// TwinCAT 3 PLC project PLC_AtoB_PlantCtrl
// ProgramVersion: 3.1.4024.0
// libraries:
//   Tc2_Standard, * (Beckhoff Automation GmbH)
//   Tc2_System, * (Beckhoff Automation GmbH)
//   Tc3_Module, * (Beckhoff Automation GmbH)
// project tree:
//   DUTs/ Udt_CM_Actuator3State.TcDUT, Udt_CM_Sensor2State.TcDUT, Udt_PlantControl_Out.TcDUT
//   GVLs/ FIO.TcGVL
//   / PlcTask.TcTTO
//   POUs/CMs/ CM_Actuator3State.TcPOU, CM_Sensor2State.TcPOU
//   POUs/ FB_PlantControl.TcPOU, MAIN.TcPOU, Prg_StateMachine.TcPOU
// real-time tasks:
//   TASK PlcTask: cycle T#10ms, priority 20, ADS port 350

CONFIGURATION PLC_AtoB_PlantCtrl
    RESOURCE PLC ON TwinCAT3
        TASK PlcTask(INTERVAL := T#10ms, PRIORITY := 20);
        PROGRAM MAIN WITH PlcTask : MAIN;
    END_RESOURCE
END_CONFIGURATION

// ---- DUTs/Udt_CM_Actuator3State.TcDUT
TYPE Udt_CM_Actuator3State :
STRUCT
	output_state1 : BOOL;
	output_state2 : BOOL;
	output_state3 : BOOL;
	
END_STRUCT
END_TYPE

// ---- DUTs/Udt_CM_Sensor2State.TcDUT
TYPE Udt_CM_Sensor2State :
STRUCT
	sensor_Input : BOOL;
	
	sensor_Output : BOOL; 
END_STRUCT
END_TYPE

// ---- DUTs/Udt_PlantControl_Out.TcDUT
TYPE Udt_PlantControl_Out :
STRUCT
	Auto_Out : BOOL;
	Manual_Out : BOOL;
	
	Startet_Out : BOOL;
	Stopped_Out : BOOL;
	Reset_Out : BOOL;
	ResetEmgStop_Out_5s :BOOL;
	
	EmgStopped_Out : BOOL;
END_STRUCT
END_TYPE

// ---- GVLs/FIO.TcGVL
{attribute 'qualified_only'}
VAR_GLOBAL
	
	bEmgStop : BOOL := TRUE; //Sensor	Bool	Emergency stop	0	TRUE
	bStart : BOOL;	//Sensor	Bool	Start	1	FALSE
	bStop : BOOL := TRUE;	//Sensor	Bool	Stop	3	TRUE
	bReset : BOOL;	//Sensor	Bool	Reset	4	FALSE
	bManual : BOOL;	//Sensor	Bool	Manual	5	TRUE
	bAuto : BOOL; 	//Sensor	Bool	Auto	6	FALSE
	
	bGreenLight : BOOL;
	bYellowLight : BOOL;
	bRedLight : BOOL;
	
	
	bSensorB : BOOL;
	bSensorA : BOOL;
	
	bEntryConveyor : BOOL;
	
	bConveyorCW : BOOL;
	bConveyorCCW : BOOL;
//Sensor	Bool	Sensor B	1	TRUE
//Sensor	Bool	Sensor A	0	TRUE

//Actuator	Bool	Roller Conveyor (4m) 1 (+)	0	FALSE
//Actuator	Bool	Roller Conveyor (4m) 1 (-)	2	FALSE
//Actuator	Bool	Entry conveyor	1	FALSE



END_VAR

// ---- POUs/MAIN.TcPOU
PROGRAM MAIN
VAR
	fbPlantControl : FB_PlantControl;
	Ctrl_data_Plant : Udt_PlantControl_Out;
	
	Ctrl_data_StateMachine :Udt_PlantControl_Out;
	
	cmSensorA : CM_Sensor2State;
	Ctrl_data_SensorA : Udt_CM_Sensor2State;
	
	cmSensorB : CM_Sensor2State;
	Ctrl_data_SensorB : Udt_CM_Sensor2State;
	
	cmConveyorEntry : CM_Actuator3State;
	Ctrl_data_ConveyorEntry : Udt_CM_Actuator3State;
	
	cmConveyorMain : CM_Actuator3State;
	Ctrl_data_ConveyorMain : Udt_CM_Actuator3State;
END_VAR

fbPlantControl(
	//Set up variables to IO here
	Auto_In := FIO.bAuto,
	Manual_In := FIO.bManual,
	
	Start_In := FIO.bStart,
	Stop_In := FIO.bStop,
	EmgStop_In := FIO.bEmgStop,
	Reset_In := FIO.bReset,
	
	Startet_Out => FIO.bGreenLight,
	Stopped_Out => FIO.bYellowLight,
	EmgStopped_Out => FIO.bRedLight,

	Ctrl_Plant := Ctrl_data_Plant
	);
	
Prg_StateMachine(
	Plant_Ctrl := Ctrl_data_Plant,
	
	cmSensor2State_sensorA := Ctrl_data_SensorA,
	cmSensor2State_sensorB := Ctrl_data_SensorB,

	cmActuator3State_ConveyorEntry :=  Ctrl_data_ConveyorEntry,
	cmActuator3State_ConveyorMain := Ctrl_data_ConveyorMain
);

cmSensorA(
	sensorInput := FIO.bSensorA,

	Ctrl_CM_Sensor2State := Ctrl_data_SensorA
	);
cmSensorB(
	sensorInput := FIO.bSensorB,

	Ctrl_CM_Sensor2State := Ctrl_data_SensorB
	);
	
cmConveyorEntry(
	output_2 => FIO.bEntryConveyor,
	
	Ctrl_CM_Actuator3State := Ctrl_data_ConveyorEntry
	);
	
cmConveyorMain(
	output_2 => FIO.bConveyorCW,
	output_3 => FIO.bConveyorCCW,
	
	Ctrl_CM_Actuator3State := Ctrl_data_ConveyorMain
	);

END_PROGRAM

// ---- POUs/FB_PlantControl.TcPOU
FUNCTION_BLOCK FB_PlantControl
VAR_INPUT
	Auto_In : BOOL;
	Manual_In : BOOL;
	
	Start_In : BOOL;
	Stop_In : BOOL;
	Reset_In : BOOL;
	
	EmgStop_In : BOOL;
	
END_VAR
VAR_OUTPUT
	Auto_Out : BOOL;
	Manual_Out : BOOL;
	
	Startet_Out : BOOL;
	Stopped_Out : BOOL;
	Reset_Out : BOOL;
	ResetEmgStop_Out_5s :BOOL;
	
	EmgStopped_Out : BOOL;
END_VAR
VAR
END_VAR
VAR_IN_OUT
	Ctrl_Plant : Udt_PlantControl_Out;
END_VAR

VAR CONSTANT
	SR_Auto: SR;
	SR_Man : SR;
	
	SR_start : SR;
	SR_Stop : SR;
	
	EmgResetTimerOff : Tc2_Standard.TON;
END_VAR

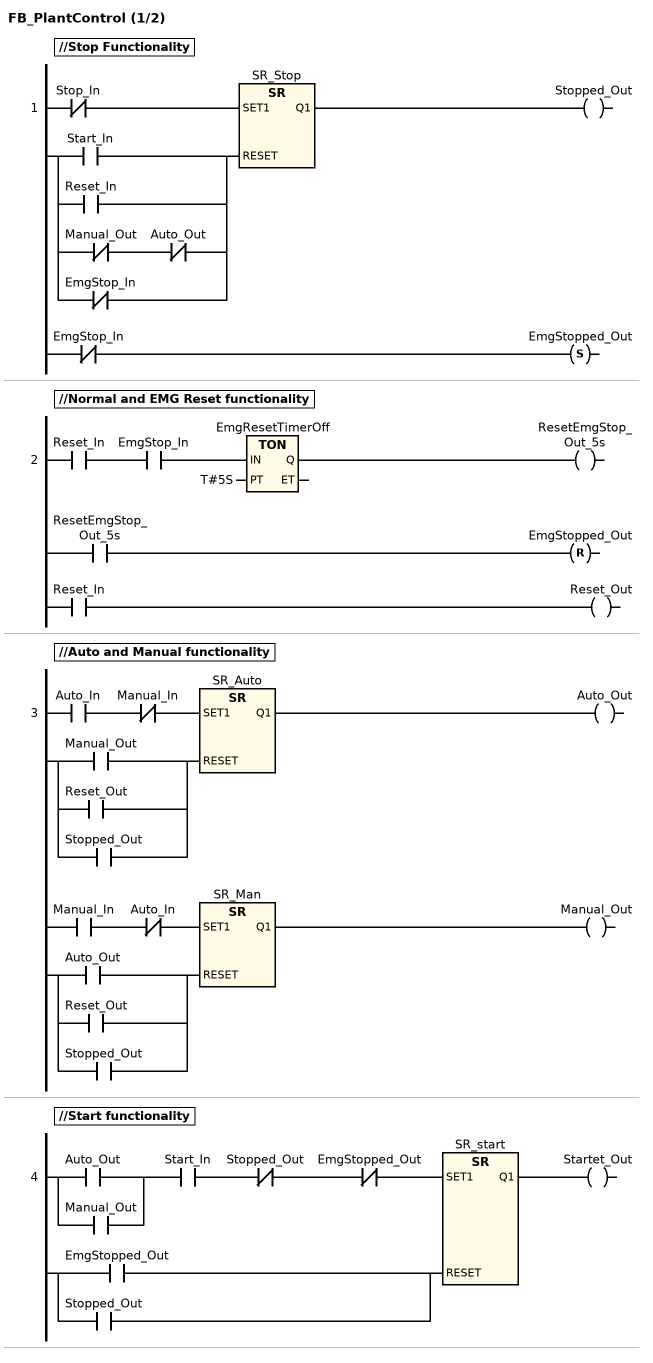
// NETWORK 1
// label: //Stop Functionality
SR_Stop(SET1 := NOT Stop_In, RESET := Start_In OR Reset_In OR NOT Manual_Out AND NOT Auto_Out OR NOT EmgStop_In); // SR
Stopped_Out := SR_Stop.Q1;
EmgStopped_Out S= NOT EmgStop_In;

// NETWORK 2
// label: //Normal and EMG Reset functionality
EmgResetTimerOff(IN := Reset_In AND EmgStop_In, PT := T#5S); // TON
ResetEmgStop_Out_5s := EmgResetTimerOff.Q;
EmgStopped_Out R= ResetEmgStop_Out_5s;
Reset_Out := Reset_In;

// NETWORK 3
// label: //Auto and Manual functionality
SR_Auto(SET1 := Auto_In AND NOT Manual_In, RESET := Manual_Out OR Reset_Out OR Stopped_Out); // SR
Auto_Out := SR_Auto.Q1;
SR_Man(SET1 := Manual_In AND NOT Auto_In, RESET := Auto_Out OR Reset_Out OR Stopped_Out); // SR
Manual_Out := SR_Man.Q1;

// NETWORK 4
// label: //Start functionality
SR_start(SET1 := (Auto_Out OR Manual_Out) AND Start_In AND NOT Stopped_Out AND NOT EmgStopped_Out, RESET := EmgStopped_Out OR Stopped_Out); // SR
Startet_Out := SR_start.Q1;

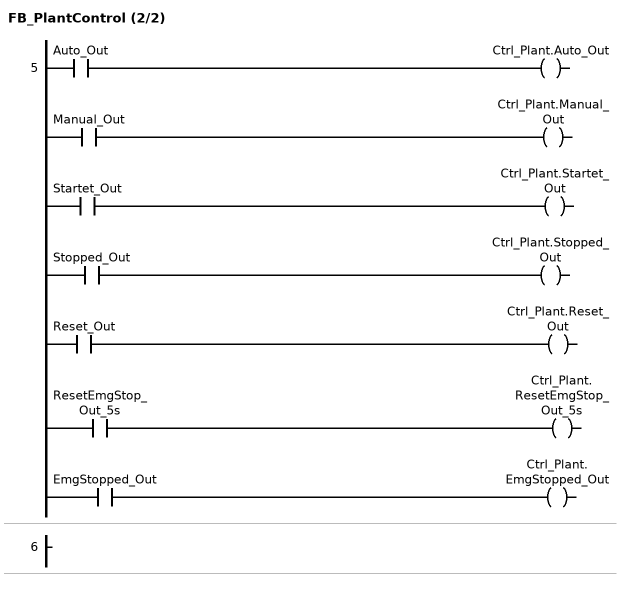
// NETWORK 5
Ctrl_Plant.Auto_Out := Auto_Out;
Ctrl_Plant.Manual_Out := Manual_Out;
Ctrl_Plant.Startet_Out := Startet_Out;
Ctrl_Plant.Stopped_Out := Stopped_Out;
Ctrl_Plant.Reset_Out := Reset_Out;
Ctrl_Plant.ResetEmgStop_Out_5s := ResetEmgStop_Out_5s;
Ctrl_Plant.EmgStopped_Out := EmgStopped_Out;

// NETWORK 6

END_FUNCTION_BLOCK

// ---- POUs/CMs/CM_Sensor2State.TcPOU
FUNCTION_BLOCK CM_Sensor2State
VAR_INPUT
	sensorInput : BOOL;
END_VAR
VAR_OUTPUT
	sensoroutput : BOOL;
END_VAR
VAR_IN_OUT
	Ctrl_CM_Sensor2State : Udt_CM_Sensor2State; 
END_VAR
VAR
END_VAR

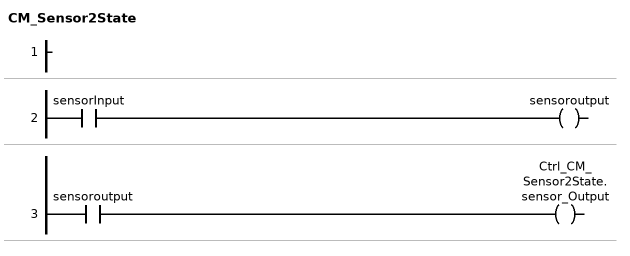
// NETWORK 1

// NETWORK 2
sensoroutput := sensorInput;

// NETWORK 3
Ctrl_CM_Sensor2State.sensor_Output := sensoroutput;

END_FUNCTION_BLOCK

// ---- POUs/CMs/CM_Actuator3State.TcPOU
FUNCTION_BLOCK CM_Actuator3State
VAR_INPUT
	
END_VAR
VAR_OUTPUT
	output_1 : BOOL;
	output_2 : BOOL;
	output_3 : BOOL;
END_VAR
VAR_IN_OUT
	Ctrl_CM_Actuator3State : Udt_CM_Actuator3State;
END_VAR
VAR
END_VAR

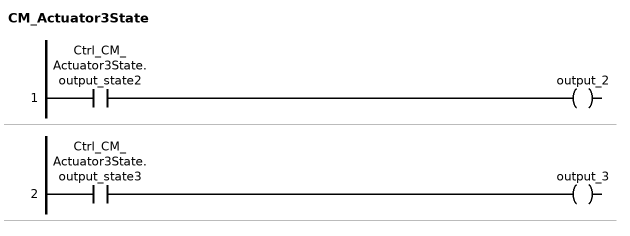
// NETWORK 1
output_2 := Ctrl_CM_Actuator3State.output_state2;

// NETWORK 2
output_3 := Ctrl_CM_Actuator3State.output_state3;

END_FUNCTION_BLOCK

// ---- POUs/Prg_StateMachine.TcPOU
PROGRAM Prg_StateMachine
VAR
	Step_0_Init : BOOL;
	Step_1 : BOOL;
	Step_2 : BOOL;
	Step_3: BOOL;
	Step_4 : BOOL;
	
	rTrigA : Tc2_Standard.R_TRIG;
	edgeA : BOOL;
	rTrigB : Tc2_Standard.R_TRIG;
	edgeB : BOOL;
END_VAR

VAR_IN_OUT
	Plant_Ctrl : Udt_PlantControl_Out;
	
	cmSensor2State_sensorA : Udt_CM_Sensor2State;
	cmSensor2State_sensorB : Udt_CM_Sensor2State;
	
	cmActuator3State_ConveyorEntry : Udt_CM_Actuator3State;
	cmActuator3State_ConveyorMain : Udt_CM_Actuator3State;
END_VAR
VAR // added by the converter: edge detectors and wires of the graphical bodies
    _w1, _w2, _w3, _w4 : BOOL;
END_VAR

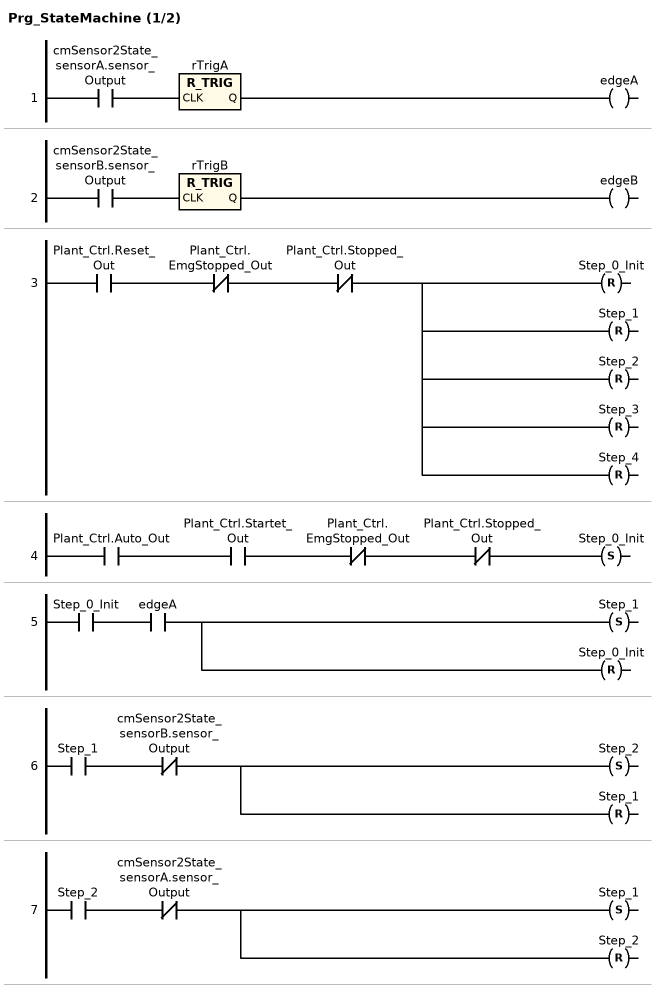
// NETWORK 1
rTrigA(CLK := cmSensor2State_sensorA.sensor_Output); // R_TRIG
edgeA := rTrigA.Q;

// NETWORK 2
rTrigB(CLK := cmSensor2State_sensorB.sensor_Output); // R_TRIG
edgeB := rTrigB.Q;

// NETWORK 3
_w1 := Plant_Ctrl.Reset_Out AND NOT Plant_Ctrl.EmgStopped_Out AND NOT Plant_Ctrl.Stopped_Out;
Step_0_Init R= _w1;
Step_1 R= _w1;
Step_2 R= _w1;
Step_3 R= _w1;
Step_4 R= _w1;

// NETWORK 4
Step_0_Init S= Plant_Ctrl.Auto_Out AND Plant_Ctrl.Startet_Out AND NOT Plant_Ctrl.EmgStopped_Out AND NOT Plant_Ctrl.Stopped_Out;

// NETWORK 5
_w2 := Step_0_Init AND edgeA;
Step_1 S= _w2;
Step_0_Init R= _w2;

// NETWORK 6
_w3 := Step_1 AND NOT cmSensor2State_sensorB.sensor_Output;
Step_2 S= _w3;
Step_1 R= _w3;

// NETWORK 7
_w4 := Step_2 AND NOT cmSensor2State_sensorA.sensor_Output;
Step_1 S= _w4;
Step_2 R= _w4;

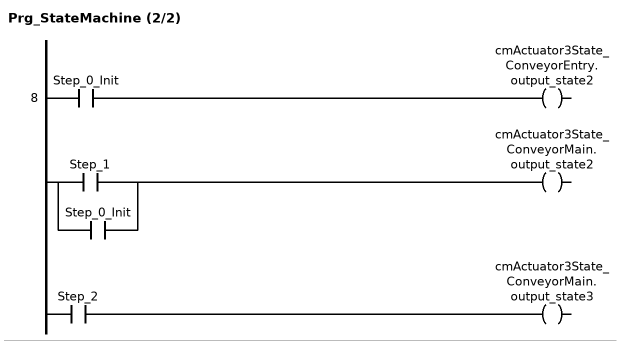
// NETWORK 8
cmActuator3State_ConveyorEntry.output_state2 := Step_0_Init;
cmActuator3State_ConveyorMain.output_state2 := Step_1 OR Step_0_Init;
cmActuator3State_ConveyorMain.output_state3 := Step_2;

END_PROGRAM
